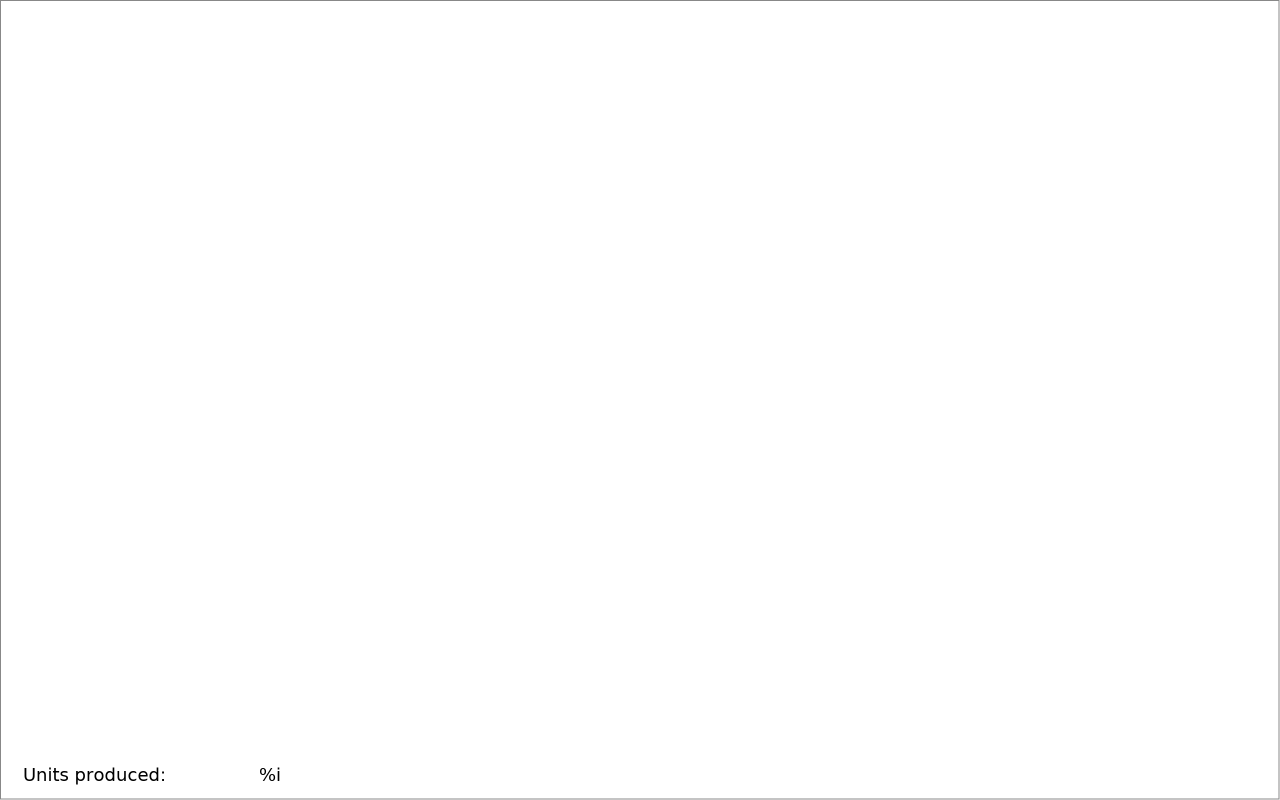
VISUALIZATION UnitsProduced  // 1280x800
VAR_IN_OUT
	nUnitsProduced : UDINT;
END_VAR
    Label (20,760 150x30), "Units produced:"
    Textfield (170,760 200x30), "%i", text variable: nUnitsProduced
END_VISUALIZATION

(* stored: Version 1.1.0.1, ProductVersion 3.1.4024.11
   Visu UnitsProduced: Id {3ccd76c5-e3be-4000-878d-db8e17feaf5e} *)
